# EPICS autosave request: iocBoot/iocelveFlowESmobile/elveFlowESmobile.req
file "elveFlow_settings.req", P=XF11ID-ES\{elveFlowOB1\}:, R=elveFlow:
file "epid.req",               P=elveFlowOB1:PID1
